(* PLC project PLCforPSM, Unknown Unnamed 1 *)
(* stored: creationDateTime 2023-03-08T11:17:00, modificationDateTime 2024-05-24T11:24:17 *)

PROGRAM b_PID4_routine
  VAR_EXTERNAL
    always_false : BOOL;  (* Always false variable *)
    Alive : BOOL;  (* Heartbeat from OpenPLC *)
    always_true : BOOL;  (* Always true variable *)
  END_VAR
  VAR
    PIT_129 : REAL;
    PIT_118 : REAL;
    LIT_125 : REAL;
    FIT_116 : REAL;
    PUMP_CH : INT := 2;
    PUMP_SPEED : INT := 0;
    KP : REAL;
    ERROR : REAL;
    INTEGRATIVE : REAL;
    SETPOINT_GEN : REAL;
    TIMEvar : REAL;
  END_VAR
  VAR_EXTERNAL
    PID_OUT : INT;  (* temporary *)
  END_VAR
  VAR
    DAQ_AI_I0 : DAQ_AI_I;
    PID_4_00 : PID_4_0;
    DAQ_AO_U_WT0 : DAQ_AO_U_WT;
  END_VAR
  VAR  (* added by the conversion: wires and edge detectors of the diagram *)
    _REAL_TO_INT90_OUT : INT;
  END_VAR

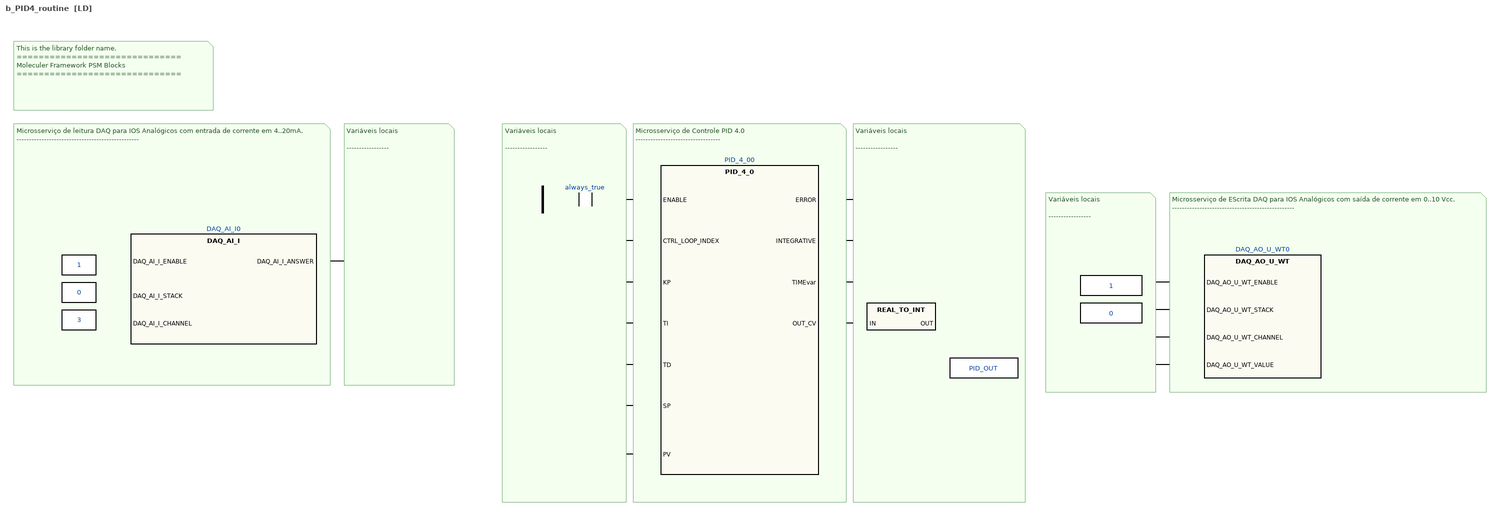
(* LD diagram, written out as Structured Text *)
(* This is the library folder name.
==============================
Moleculer Framework PSM Blocks
============================== *)
(* Microsserviço de leitura DAQ para IOS Analógicos com entrada de corrente em 4..20mA.
------------------------------------------------- *)
(* Variáveis locais

----------------- *)
(* Microsserviço de Controle PID 4.0
---------------------------------- *)
(* Variáveis locais

----------------- *)
(* Variáveis locais

----------------- *)
(* Variáveis locais

----------------- *)
(* Microsserviço de EScrita DAQ para IOS Analógicos com saída de corrente em 0..10 Vcc.
------------------------------------------------- *)
DAQ_AI_I0(DAQ_AI_I_ENABLE := 1, DAQ_AI_I_STACK := 0, DAQ_AI_I_CHANNEL := 3);
LIT_125 := DAQ_AI_I0.DAQ_AI_I_ANSWER;
PID_4_00(ENABLE := always_true, CTRL_LOOP_INDEX := 1, KP := 30.0, TI := 5.0, TD := 0.01, SP := 50.0, PV := LIT_125);
_REAL_TO_INT90_OUT := REAL_TO_INT(PID_4_00.OUT_CV);
PUMP_SPEED := _REAL_TO_INT90_OUT;
INTEGRATIVE := PID_4_00.INTEGRATIVE;
TIMEvar := PID_4_00.TIMEvar;
ERROR := PID_4_00.ERROR;
PID_OUT := _REAL_TO_INT90_OUT;
DAQ_AO_U_WT0(DAQ_AO_U_WT_ENABLE := 1, DAQ_AO_U_WT_STACK := 0, DAQ_AO_U_WT_CHANNEL := 2, DAQ_AO_U_WT_VALUE := PUMP_SPEED);
END_PROGRAM

PROGRAM a_Main_routine
  VAR_EXTERNAL
    Alive : BOOL;  (* Heartbeat from OpenPLC *)
  END_VAR
  VAR
    TON0 : TON;
    TON1 : TON;
  END_VAR
  VAR_EXTERNAL
    always_false : BOOL;
    always_true : BOOL;
    DAQ_AI_I_ch1 : REAL;  (* Global Variable for general use *)
    DAQ_AI_I_ch2 : REAL;  (* Global Variable for general use (LIT 125) *)
    DAQ_AI_I_ch3 : REAL;  (* Global Variable for general use *)
    DAQ_AI_I_ch4 : REAL;  (* Global Variable for general use *)
  END_VAR

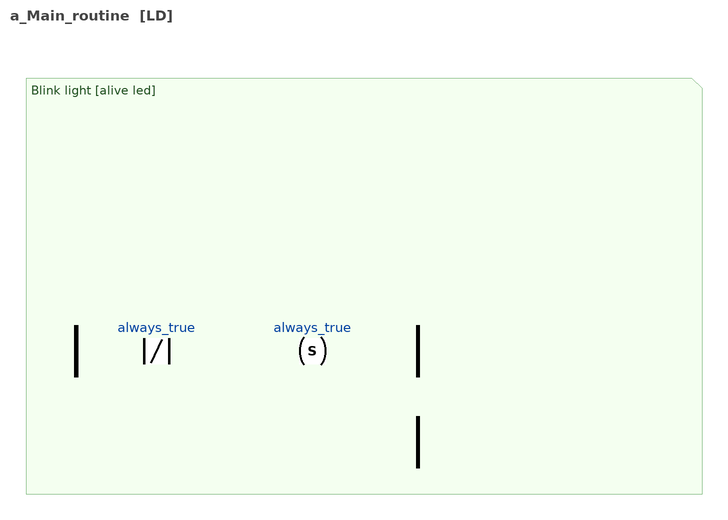
(* LD diagram, written out as Structured Text *)
(* Blink light [alive led] *)
TON0(IN := NOT TON1.q, PT := T#5000ms);
Alive := TON0.Q;
IF always_false THEN always_false := FALSE; END_IF;
IF NOT always_true THEN always_true := TRUE; END_IF;
TON1(IN := TON0.Q, PT := T#5000ms);
END_PROGRAM

CONFIGURATION Config0
  RESOURCE Res0 ON PLC
    VAR_GLOBAL
      always_false AT %QX0.0 : BOOL := 0;  (* Always false variable *)
      always_true AT %QX0.1 : BOOL := 1;  (* Always true variable *)
      Alive AT %QX0.2 : BOOL := 0;  (* Heartbeat from OpenPLC *)
      DAQ_AI_I_ENABLE_PSM AT %QX1.0 : BOOL := 0;  (* # Enable DAQ reading to PSM (%QX1.0) *)
      DAQ_AI_I_STACK_PSM AT %QW14 : INT := 0;  (* # Stack for Megaind Board [0..7] (%QW14) *)
      DAQ_AI_I_CHANNEL_PSM AT %QW15 : INT := 0;  (* # Channel number for Megaind board [0..3] (%QW15) *)
      DAQ_AI_I_PSM AT %IW20 : INT := 0;  (* # Analog Input Current from PSM (int) [x100] (%IW20) *)
      DAQ_AI_I_ch1 : REAL := 0;  (* Global Variable for general use *)
      DAQ_AI_I_ch2 : REAL := 0;  (* Global Variable for general use *)
      DAQ_AI_I_ch3 : REAL := 0;  (* Global Variable for general use *)
      DAQ_AI_I_ch4 : REAL := 0;  (* Global Variable for general use *)
      DAQ_AO_U_WT_ENABLE_PSM AT %QX0.3 : BOOL := 0;  (* # Enable DAQ writing to PSM (%QX0.3) *)
      DAQ_AO_U_WT_STACK_PSM AT %QW2 : INT := 0;  (* # Stack for Megaind Board [0..7] (%QW2) *)
      DAQ_AO_U_WT_CHANNEL_PSM AT %QW3 : INT := 0;  (* # Channel number for Megaind board [0..3] (%QW3) *)
      DAQ_AO_U_WT_VALUE_PSM AT %QW4 : INT := 0;  (* # Output Value for Megaind board [0..100] (%QW4) *)
      DAQ_AO_U_RD_ENABLE_PSM AT %QX0.4 : BOOL := 0;  (* # Enable DAQ writing to PSM (%QX0.4) *)
      DAQ_AO_U_RD_STACK_PSM AT %QW5 : INT := 0;  (* # Stack for Megaind Board [0..7] (%QW5) *)
      DAQ_AO_U_RD_CHANNEL_PSM AT %QW6 : INT := 0;  (* # Channel number for Megaind board [1..4] (%QW6) *)
      DAQ_AO_U_RD_PSM AT %IW21 : INT := 0;  (* # Analog output voltage from PSM (int) [x100] (%IW21) *)
      DAQ_AI_U_ENABLE_PSM AT %QX0.5 : BOOL := 0;  (* # Enable DAQ reading to PSM (%QX0.5) *)
      DAQ_AI_U_STACK_PSM AT %QW7 : INT := 0;  (* # Stack for Megaind Board [0..7] (%QW7) *)
      DAQ_AI_U_CHANNEL_PSM AT %QW8 : INT := 0;  (* # Channel number for Megaind board [0..3] (%QW8) *)
      DAQ_AI_U_PSM AT %IW22 : INT := 0;  (* # Analog output voltage from PSM (int) [x100] (%IW22) *)
      DAQ_AO_I_WT_ENABLE_PSM AT %QX0.6 : BOOL := 0;  (* # Enable DAQ writing to PSM (%QX0.6) *)
      DAQ_AO_I_WT_STACK_PSM AT %QW9 : INT := 0;  (* # Stack for Megaind Board [0..7] (%QW9) *)
      DAQ_AO_I_WT_CHANNEL_PSM AT %QW10 : INT := 0;  (* # Channel number for Megaind board [0..3] (%QW10) *)
      DAQ_AO_I_WT_VALUE_PSM AT %QW11 : INT := 0;  (* # Output Value for Megaind board [0..100] (%QW11) *)
      DAQ_AO_I_RD_ENABLE_PSM AT %QX0.7 : BOOL := 0;  (* # Enable DAQ reading to PSM (%QX0.7) *)
      DAQ_AO_I_RD_STACK_PSM AT %QW12 : INT := 0;  (* # Stack for Megaind Board [0..7] (%QW12) *)
      DAQ_AO_I_RD_CHANNEL_PSM AT %QW13 : INT := 0;  (* # Channel number for Megaind board [1..4] (%QW13) *)
      DAQ_AO_I_RD_PSM AT %IW23 : INT := 0;  (* # Analog output current from PSM (int) [x100] (%IW23) *)
      DAQ_AO_OD_WT_ENABLE_PSM AT %QX1.1 : BOOL := 0;  (* # Enable DAQ writing to PSM (%QX1.1) *)
      DAQ_AO_OD_WT_STACK_PSM AT %QW16 : INT := 0;  (* # Stack for Megaind Board [0..7] (%QW16) *)
      DAQ_AO_OD_WT_CHANNEL_PSM AT %QW17 : INT := 0;  (* # Channel number for Megaind board [0..3] (%QW17) *)
      DAQ_AO_OD_WT_VALUE_PSM AT %QW18 : INT := 0;  (* # Output Value for Megaind board [0..100] (%QW18) *)
      DAQ_AO_OD_RD_ENABLE_PSM AT %QX1.2 : BOOL := 0;  (* # Enable DAQ writing to PSM (%QX1.2) *)
      DAQ_AO_OD_RD_STACK_PSM AT %QW19 : INT := 0;  (* # Stack for Megaind Board [0..7] (%QW19) *)
      DAQ_AO_OD_RD_CHANNEL_PSM AT %QW20 : INT := 0;  (* # Channel number for Megaind board [0..3] (%QW20) *)
      DAQ_AO_OD_RD_PSM AT %IW24 : INT := 0;  (* # Analog output voltage from PSM (int) [x100] (%IW24) *)
      DAQ_DI_OPTO_ENABLE_PSM AT %QX1.3 : BOOL := 0;  (* # Enable DAQ writing to PSM (%QX1.3) *)
      DAQ_DI_OPTO_STACK_PSM AT %QW21 : INT := 0;  (* # Stack for Megaind Board [0..7] (%QW21) *)
      DAQ_DI_OPTO_CHANNEL_PSM AT %QW22 : INT := 0;  (* # Channel number for Megaind board [0..3] (%QW22) *)
      DAQ_DI_OPTO_PSM AT %IW25 : INT := 0;  (* # Digital Input from PSM (int) [x100] (%IW25) *)
      PID4_ENABLED_PSM AT %QX1.4 : BOOL := 0;  (* PID4 - Enable PID 4.0 to PSM (%QW1.4) *)
      CTRL_LOOP_INDEX_PSM AT %QW23 : INT := 0;  (* PID4 - Unique Integer Number to define the control loop (%QW41) *)
      KP_PSM AT %QW24 : INT := 0;  (* PID4 - KP to PSM (x10) (%QW24) *)
      TI_PSM AT %QW25 : INT := 0;  (* PID4 - (PID4 - 10) I=xx; Ti=P/I [To reduce its installment, make Ti higher than 1.0] (%QW25) *)
      TD_PSM AT %QW26 : INT := 0;  (* PID4 - (x10) D=xx; Td=D/P [To reduce its installment, make Ti smaller than 1.0] (%QW26) *)
      PV_PSM AT %QW27 : INT := 0;  (* PID4 - (x10) PV to PSM (%QW27) *)
      SP_PSM AT %QW28 : INT := 0;  (* PID4 - (x10) Setpoint to PSM (%QW28) *)
      ERROR_PSM AT %IW26 : INT := 0;  (* PID4 - Erro variable from PSM (%IW26) *)
      INTEGRATIVE_PSM AT %IW27 : INT := 0;  (* PID4 - Integrative variable from PSM (%IW27) *)
      TIMEpsm AT %IW28 : INT := 0;  (* PID4 - Time Variable from PSM (%IW28) *)
      OUT_CV_PSM AT %IW29 : INT := 0;  (* PID4 - Control Variable from PSM (%IW29) *)
      PID_OUT AT %QW29 : INT := 0;  (* temporary *)
    END_VAR
    TASK Main(INTERVAL := T#100ms, PRIORITY := 1);
    PROGRAM instance00 WITH Main : a_Main_routine;
    PROGRAM instance01 WITH Main : b_PID4_routine;
  END_RESOURCE
END_CONFIGURATION
